// TIA Portal project "production line" (V17)
// Vorlageprojekt für das Buch mit Zielsystem S7-1200

(* hardware
DEVICE "S7-1200-Station_1"  S7-1200 Station
   slot 0: "Baugruppenträger_0"  Rack  V1.0
   slot 1: "PLC_1"  CPU 1211C DC/DC/DC  6ES7 211-1AE40-0XB0  V4.1
*)

// ===== PLC "PLC_1"  CPU 1211C DC/DC/DC =====

VAR_GLOBAL   // PLC tag table "Standard-Variablentabelle"
   "lids at entry" AT %I0.0 : Bool;
   "lid center busy" AT %I0.1 : Bool;
   "lid center error" AT %I0.2 : Bool;
   "lid at exit" AT %I0.3 : Bool;
   "base at entry" AT %I0.4 : Bool;
   "base center busy" AT %I0.5 : Bool;
   "base center error" AT %I0.6 : Bool;
   "base at exit" AT %I0.7 : Bool;
   "FACTORY io run" AT %I1.0 : Bool;
   "lid r conv" AT %Q0.0 : Bool;
   "produce lids lc" AT %Q0.1 : Bool;
   "start lc" AT %Q0.2 : Bool;
   "reset lc" AT %Q0.3 : Bool;
   "stop lc" AT %Q0.4 : Bool;
   "lid exit conv1" AT %Q0.5 : Bool;
   "liv exit conv2" AT %Q0.6 : Bool;
   "base r conv" AT %Q0.7 : Bool;
   "produce lids bc" AT %Q1.0 : Bool;
   "start bc" AT %Q1.1 : Bool;
   "reset bc" AT %Q1.2 : Bool;
   "stop bc" AT %Q1.3 : Bool;
   "base exit conv1" AT %Q1.4 : Bool;
   "base exit conv2" AT %Q1.5 : Bool;
   "exit conv" AT %Q1.6 : Bool;
   "lid counter" AT %QD30 : DInt;
   "base counter" AT %QD34 : DInt;
   "Tag_1" AT %M0.0 : Bool;
   "start" AT %I1.1 : Bool;
   "reset lid" AT %M1.0 : Bool;
   "reset base" AT %M1.1 : Bool;
   "Tag_2" AT %M0.1 : Bool;
END_VAR

DATA_BLOCK "modes"   // DB2
{ S7_Optimized_Access := 'TRUE' }
VERSION : 0.1
   VAR
      "stop mode" : Bool;
      "start mode" : Bool;
      "reset mode" : Bool;
   END_VAR
BEGIN
END_DATA_BLOCK

// folder: System blocks/Program resources

DATA_BLOCK "count lid"   // DB1
{ S7_Optimized_Access := 'TRUE' }
AUTHOR : Simatic
FAMILY : IEC
NAME : CNTR
VERSION : 1.0
// stored: InstanceOfName IEC_COUNTER
"IEC_COUNTER"
BEGIN
END_DATA_BLOCK

DATA_BLOCK "count base"   // DB3
{ S7_Optimized_Access := 'TRUE' }
AUTHOR : Simatic
FAMILY : IEC
NAME : CNTR
VERSION : 1.0
// stored: InstanceOfName IEC_COUNTER
"IEC_COUNTER"
BEGIN
END_DATA_BLOCK

// folder: (top level)

FUNCTION "1 operation modes" : Void   // FC1, LAD
{ S7_Optimized_Access := 'TRUE' }
VERSION : 0.1
BEGIN

REGION Network 1: start mode
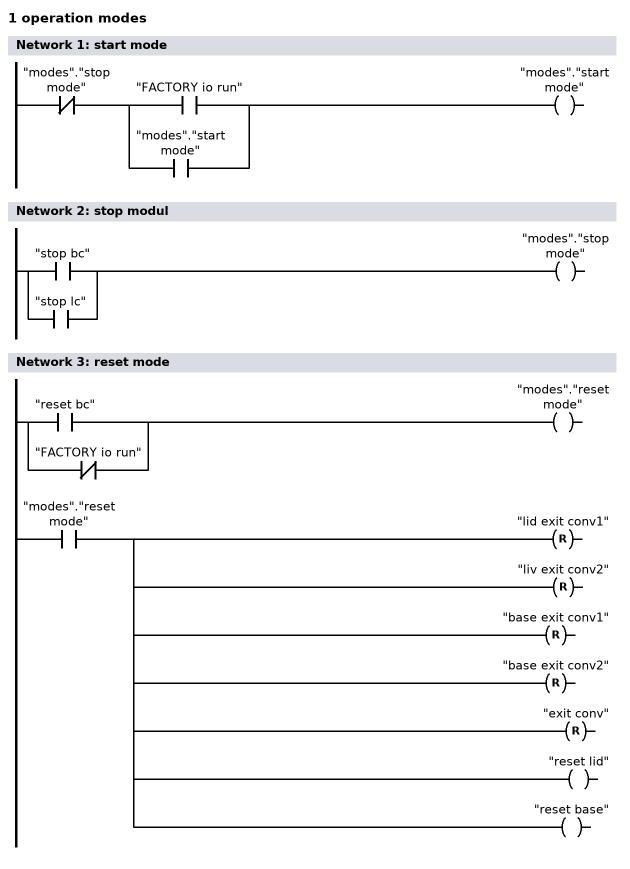
   RUNG wire#powerrail
      I_Contact( "modes"."stop mode" )
      wire#w1
      Contact( "FACTORY io run" )
      wire#w2
      Coil( "modes"."start mode" )
   END_RUNG
   RUNG wire#w1
      Contact( "modes"."start mode" )
   END_RUNG wire#w2
   // the same network as SCL:
   "modes"."start mode" := NOT "modes"."stop mode" AND ("FACTORY io run" OR "modes"."start mode");
END_REGION

REGION Network 2: stop modul
   RUNG wire#powerrail
      Contact( "stop bc" )
      wire#w1
      Coil( "modes"."stop mode" )
   END_RUNG
   RUNG wire#powerrail
      Contact( "stop lc" )
   END_RUNG wire#w1
   // the same network as SCL:
   "modes"."stop mode" := "stop bc" OR "stop lc";
END_REGION

REGION Network 3: reset mode
   RUNG wire#powerrail
      Contact( "reset bc" )
      wire#w1
      Coil( "modes"."reset mode" )
   END_RUNG
   RUNG wire#powerrail
      I_Contact( "FACTORY io run" )
   END_RUNG wire#w1
   RUNG wire#powerrail
      Contact( "modes"."reset mode" )
      wire#w2
      R_Coil( "lid exit conv1" )
   END_RUNG
   RUNG wire#w2
      R_Coil( "liv exit conv2" )
   END_RUNG
   RUNG wire#w2
      R_Coil( "base exit conv1" )
   END_RUNG
   RUNG wire#w2
      R_Coil( "base exit conv2" )
   END_RUNG
   RUNG wire#w2
      R_Coil( "exit conv" )
   END_RUNG
   RUNG wire#w2
      Coil( "reset lid" )
   END_RUNG
   RUNG wire#w2
      Coil( "reset base" )
   END_RUNG
   // the same network as SCL:
   "modes"."reset mode" := "reset bc" OR NOT "FACTORY io run";
   IF "modes"."reset mode" THEN
       "lid exit conv1" := FALSE;
       "liv exit conv2" := FALSE;
       "base exit conv1" := FALSE;
       "base exit conv2" := FALSE;
       "exit conv" := FALSE;
   END_IF;
   "reset lid" := "modes"."reset mode";
   "reset base" := "modes"."reset mode";
END_REGION
END_FUNCTION

FUNCTION "2 step definition" : Void   // FC2, LAD
{ S7_Optimized_Access := 'TRUE' }
VERSION : 0.1
BEGIN

REGION Network 1
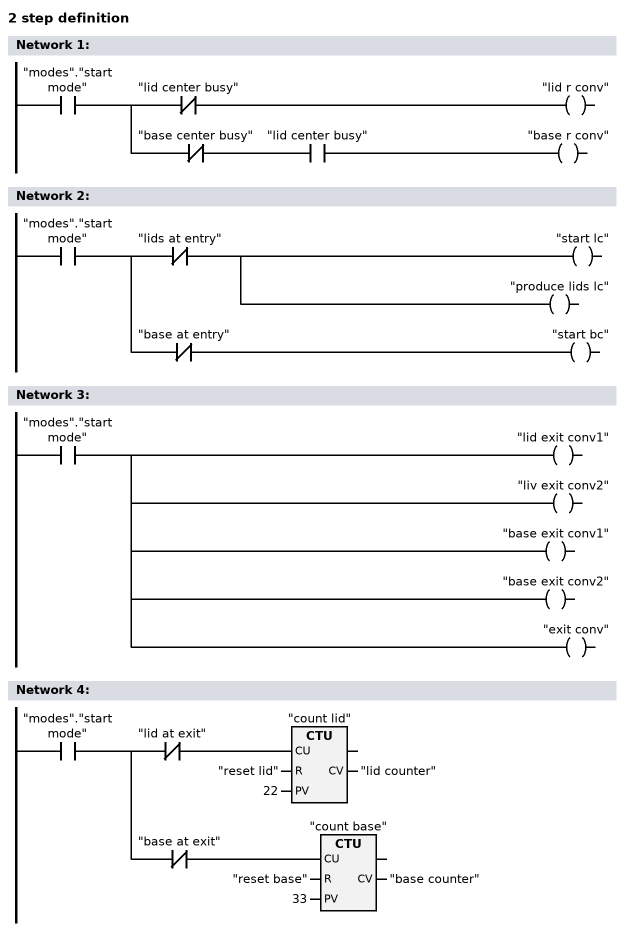
   RUNG wire#powerrail
      Contact( "modes"."start mode" )
      wire#w1
      I_Contact( "lid center busy" )
      Coil( "lid r conv" )
   END_RUNG
   RUNG wire#w1
      I_Contact( "base center busy" )
      Contact( "lid center busy" )
      Coil( "base r conv" )
   END_RUNG
   // the same network as SCL:
   "lid r conv" := "modes"."start mode" AND NOT "lid center busy";
   "base r conv" := "modes"."start mode" AND NOT "base center busy" AND "lid center busy";
END_REGION

REGION Network 2
   RUNG wire#powerrail
      Contact( "modes"."start mode" )
      wire#w1
      I_Contact( "lids at entry" )
      wire#w2
      Coil( "start lc" )
   END_RUNG
   RUNG wire#w2
      Coil( "produce lids lc" )
   END_RUNG
   RUNG wire#w1
      I_Contact( "base at entry" )
      Coil( "start bc" )
   END_RUNG
   // the same network as SCL:
   "start lc" := "modes"."start mode" AND NOT "lids at entry";
   "produce lids lc" := "start lc";
   "start bc" := "modes"."start mode" AND NOT "base at entry";
END_REGION

REGION Network 3
   RUNG wire#powerrail
      Contact( "modes"."start mode" )
      wire#w1
      Coil( "lid exit conv1" )
   END_RUNG
   RUNG wire#w1
      Coil( "liv exit conv2" )
   END_RUNG
   RUNG wire#w1
      Coil( "base exit conv1" )
   END_RUNG
   RUNG wire#w1
      Coil( "base exit conv2" )
   END_RUNG
   RUNG wire#w1
      Coil( "exit conv" )
   END_RUNG
   // the same network as SCL:
   "lid exit conv1" := "modes"."start mode";
   "liv exit conv2" := "modes"."start mode";
   "base exit conv1" := "modes"."start mode";
   "base exit conv2" := "modes"."start mode";
   "exit conv" := "modes"."start mode";
END_REGION

REGION Network 4
   "count lid".CTU(CU := "modes"."start mode" AND NOT "lid at exit",
                   R := "reset lid",
                   PV := 22,
                   CV => "lid counter");
   "count base".CTU(CU := "modes"."start mode" AND NOT "base at exit",
                    R := "reset base",
                    PV := 33,
                    CV => "base counter");
END_REGION
END_FUNCTION

FUNCTION "MHJ-PLC-Lab-Function-S71200" : Void   // FC9000, SCL
{ S7_Optimized_Access := 'TRUE' }
VERSION : 0.1
   VAR_TEMP
      rdTimeReturn : Int;
      outputTime : DTL;
      SyncVal : Byte;
      forVal : Int;
      forVal_2 : Int;
      Value : Byte;
   END_VAR
   VAR CONSTANT
      CompVal : Byte := 16#34;
      Value_01 : Byte := 16#11;
      Value_01_DW : DWord := 16#A165_D992;
      Value_02_DW : DWord := 16#58BE_4401;
   END_VAR
BEGIN

   #Value:=PEEK(area := 16#82,
        dbNumber := 0,
        byteOffset := 511);
   #Value := #Value + 1;

   POKE(area := 16#82,
        dbNumber := 0,
        byteOffset := 511,
        value := #Value);

   POKE(area:=16#81,
        dbNumber:=0,
        byteOffset:=1016,
        value:=#Value_01_DW);
   POKE(area := 16#81,
        dbNumber := 0,
        byteOffset := 1020,
        value := #Value_02_DW);

   POKE(area := 16#81,
        dbNumber := 0,
        byteOffset := 511,
        value := B#16#00);

   FOR #forVal := 0 TO 120 DO
       FOR #forVal_2:=0 TO 10 DO
           #rdTimeReturn:=RD_SYS_T(#outputTime);
           #rdTimeReturn := WR_SYS_T(#outputTime);
           #rdTimeReturn := RD_SYS_T(#outputTime);
           #rdTimeReturn := WR_SYS_T(#outputTime);
       END_FOR;
       #SyncVal:= PEEK(area := 16#81,
                      dbNumber := 0,
                      byteOffset := 511);
       IF #SyncVal = #CompVal THEN
          GOTO M_1;
       END_IF;
   END_FOR;
   RETURN;

   M_1:
   POKE(area := 16#81,
        dbNumber := 0,
        byteOffset := 511,
        value := B#16#0);
END_FUNCTION

ORGANIZATION_BLOCK "Main"   // OB1, FBD, ProgramCycle
TITLE = "Main Program Sweep (Cycle)"
{ S7_Optimized_Access := 'TRUE' }
VERSION : 0.1
   VAR_INPUT
      Initial_Call : Bool;   // Initial call of this OB
      Remanence : Bool;   // =True, if remanent data are available
   END_VAR
BEGIN

REGION Network 1: Konnektierungsbaustein für PLC-Lab
   // Im Netzwerk 1 wird der Konnektierungsbaustein für PLC-Lab aufgerufen.
   // Dieser Aufruf darf nicht entfernt werden!
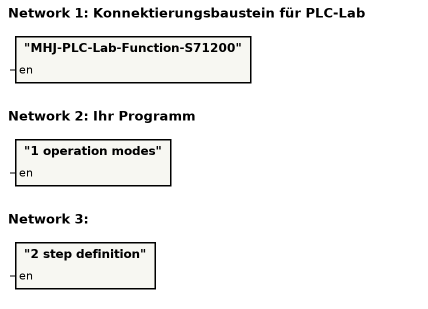
   "MHJ-PLC-Lab-Function-S71200"();
END_REGION

REGION Network 2: Ihr Programm
   // Schreiben Sie ab Netzwerk 2 Ihr Programm
   "1 operation modes"();
END_REGION

REGION Network 3
   "2 step definition"();
END_REGION
END_ORGANIZATION_BLOCK